{attribute addProperty BoxType "AMI8000-0000-0016"}
{attribute addProperty Id "WcStateAT %I*BIT10.1250InputToggleAT %I*BIT10.1250"}
{attribute addProperty CRC "2560941941"}
{attribute addProperty SizeInBites "2"}
{attribute addProperty SizeInBytes "0.25"}
TYPE WcState_98A4DF75 :
STRUCT
	{attribute addProperty Name "WcState"}
	WcState AT %I* : BIT;
	{attribute addProperty Name "InputToggle"}
	InputToggle AT %I* : BIT;
END_STRUCT
END_TYPE

(* stored: Version 1.2.0.0, ProductVersion 3.1.4024.9
   DUT WcState_98A4DF75: Id {ba89822a-3432-42f1-b4ca-7014821b2261} *)
